PROGRAM TestRunner
VAR
 	packml_test_suite : PackMLTestSuite;
	unit_mode : MockUnitMode;
END_VAR

TcUnit.Run();

END_PROGRAM

(* stored: Version 1.1.0.1
   POU TestRunner: Id {9987c82e-34e1-4813-9836-1a87627bcb36}, SpecialFunc None *)
